FUNCTION_BLOCK Machine EXTENDS FB_PackML_BaseModule
VAR
	Infeed	: Infeed  := (Name := 'Infeed');
	Outfeed : Outfeed := (Name := 'Outfeed');
END_VAR

// Automatically enables and disables HMI control based on the PackML mode
METHOD PROTECTED HMIPermissions

// This method is called cyclically by CyclicLogic()
AllowHMIControl(TRUE);
END_METHOD

// Basic module initialization logic
METHOD PROTECTED Initialize : BOOL;
VAR
	i						 : UDINT;
	varInfo					 : __SYSTEM.VAR_INFO;
	AllSubUnitsInitialized	 : BOOL := TRUE;
	AllComponentsInitialized : BOOL := TRUE;
END_VAR

// This method is called by CyclicLogic() as required
Initialize := FALSE;
CASE DescendantSequenceState OF
	0:
		RegisterSubmodule(SubModule := Infeed);
		RegisterSubmodule(SubModule := Outfeed);
		DescendantSequenceState := DescendantSequenceState + 10;

	10:
		IF SUPER^.Initialize() THEN
			DescendantSequenceState := DescendantSequenceState + 10;
		END_IF

	20:
		Initialize := TRUE;
END_CASE
END_METHOD

END_FUNCTION_BLOCK

(* stored: Version 1.1.0.1, ProductVersion 3.1.4024.12
   POU Machine: Id {51700833-d554-46cc-805c-c30409d4d74a}, SpecialFunc None
   Method HMIPermissions: Id {c36b9406-3764-4aab-a1ca-5f6b6029257d}
   Method Initialize: Id {4836559d-cfa2-4829-b680-3f2f6c73e335} *)
